{attribute 'linkalways'} 
{attribute 'no_explicit_call' := 'This FB is a CLASS and must be accessed using methods or properties'}
{attribute 'enable_dynamic_creation'}
FUNCTION_BLOCK SubscriberCollection
VAR
	collection : Collection;
END_VAR

PROPERTY PUBLIC Count : UDINT
GET
Count := collection.Count;
END_GET
END_PROPERTY

METHOD PUBLIC GetByIndex : I_Subscriber
VAR_INPUT
	Index : UDINT;
END_VAR
VAR
	subscriber : I_Subscriber;
END_VAR
IF __QUERYINTERFACE(collection.GetByIndex(Index),subscriber) THEN
	GetByIndex := subscriber;
END_IF
END_METHOD

METHOD PUBLIC Insert
VAR_INPUT
	Subscriber : I_Subscriber;
END_VAR
VAR
	collectable : I_Collectable;
END_VAR
IF __QUERYINTERFACE(Subscriber,collectable) THEN
	collection.Insert(collectable);
END_IF
END_METHOD

METHOD Remove : BOOL
VAR_INPUT
	Subscriber : I_Subscriber;
END_VAR
VAR
	collectable : I_Collectable;
END_VAR
IF __QUERYINTERFACE(Subscriber,collectable) THEN
	collection.Remove(collectable);
END_IF
END_METHOD

END_FUNCTION_BLOCK

(* stored: Version 1.1.0.1, ProductVersion 3.1.4024.12
   POU SubscriberCollection: Id {d917c827-2396-0484-2b8f-82bcb6cde2f1}, SpecialFunc None
   Property Count: Id {a9dbebc5-b868-073a-2389-984c104d3d63}
   Get Get: Id {7af500d7-4fe2-0796-2c4c-da33afde5a62}
   Method GetByIndex: Id {5b0c3edb-54d1-036d-1bd9-0370ddf07d37}
   Method Insert: Id {2b8cee3c-488f-0e91-36eb-37f4104f5bf5}
   Method Remove: Id {c85bf324-887c-0a41-25a5-3804d94c863b} *)
